{attribute 'GeneratedUsingTerminal: EL9576-0000-0019'}
{attribute addProperty BoxType "EL9576-0000-0019"}
{attribute addProperty Id "BCT_InputsAT %I*BCT_Inputs_4B98789517WcStateAT %I*WcState_9091E0EB2InfoDataAT %I*InfoData_94A18F5E2"}
{attribute addProperty CRC "3850431520"}
{attribute addProperty Size "21"}
TYPE EL9576_E580EC20 EXTENDS EtcSlaveTerminalBase_947E5A46 :
STRUCT
	{attribute addProperty Name "BCT_Inputs"}
	BCT_Inputs : BCT_Inputs_4B987895;
	{attribute addProperty Name "WcState"}
	WcState : WcState_9091E0EB;
	{attribute addProperty Name "InfoData"}
	InfoData : InfoData_94A18F5E;
END_STRUCT
END_TYPE

(* stored: Version 1.2.0.0, ProductVersion 3.1.4024.9
   DUT EL9576_E580EC20: Id {8aea4eed-57a1-4d70-a1c6-9d88300b2210} *)
